{attribute 'qualified_only'}
{attribute 'strict'}
TYPE E_Z3_Step :
(
	(* special steps *)
	NoStep := -32767,		// nessuno step
	Unknown := -32000,		// step sconosciuto
	
	(* Error steps *)
	NeOrError := -990,		// non abilitata o in errore
	Recovering := -980,		// azzeramento errori
		
	(* Stop *)
	Stop := 0,				// S0, stop
	
	(* Cycle *)
	Ready := 100,			// S1, pronto a ricevere pezzo
	MoveToMill := 120,		// S2, avanza il nastro fino alla fresa
	Milling := 140,			// S3, lavorazione con la fresa
	WaitZ4Ready := 160,		// S4, attende che Z4 sia ready
	MoveToZ4 := 180,		// S5, avanza il nastro fino a Z4

	Done := 800,			// Ciclo concluso
	
	(* Stopping *)
	Stopping := 900	
);
END_TYPE
//  NoStep = '-32767'
//  Unknown = '-32000'
//  NeOrError = '-990'
//  Recovering = '-980'

(* stored: Version 1.1.0.1
   EnumerationTextList E_Z3_Step: Id {44e142bc-df9f-0d0f-2ab2-ba5dee166e6e} *)
